Fanuc KAREL source: kt00720.KL

-- PROVISIONAL review KL for V1013-1; original PC SHA256 6a4152dd0338d3519199dcc481653e1ace86f91369a2596d1c98f70a8a5eb0b4
-- Incomplete behavior may be omitted. Consult companion uncertainty JSON. Do not deploy.
PROGRAM KT00720
%NOLOCKGROUP
VAR
  OUT : BOOLEAN
-- UNRESOLVED_DECL P1 type=000102
-- UNRESOLVED_DECL P2 type=000102
BEGIN
  -- UNRESOLVED_PC offsets 5-20; opcodes 2E,22,32,35
  -- UNRESOLVED_PC offsets 25-40; opcodes 2E,22,32,35
  -- UNRESOLVED_PC offsets 45-60; opcodes 2E,22,32,35
  -- UNRESOLVED_PC offsets 65-80; opcodes 2E,22,32,35
  -- UNRESOLVED_PC offsets 85-100; opcodes 22,63,23
  -- UNRESOLVED_PC offsets 105-109; opcodes 7F
END KT00720
